TYPE "Thickness_PersData"
VERSION : 0.1
// Block: Thickness_PersData
   STRUCT
      Measure : Struct
         BypassON : Bool;
         ID : DInt;
         Last_TriggerPosition : LReal;
         AverageSum : LReal;
         OutOfRange_Counter : Int;
         InRange_Counter : Int;
         Buffer : Array[1..THICKNESS_CHECK__BUFFER_ITEMS] of Thickness_Measure_Item;
      END_STRUCT;
      MES_Record : Thickness_Measure_Item;
   END_STRUCT;

END_TYPE
